Yaskawa INFORM job: pos_z_2.JBI

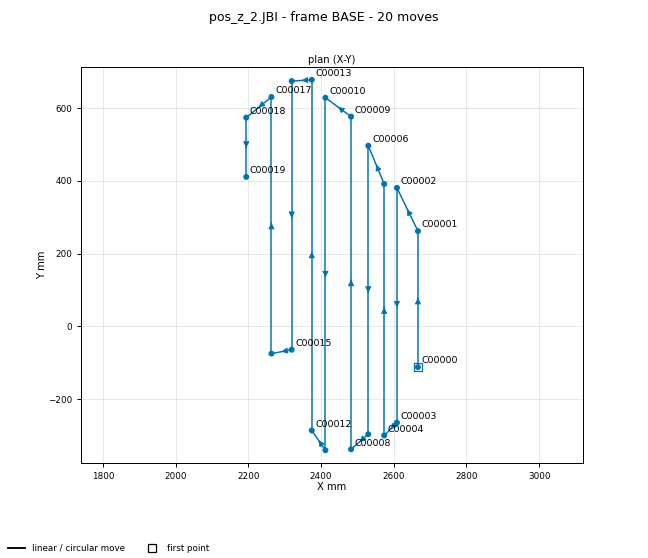
[picture p0: tool path of pos_z_2.JBI in frame BASE, 20 of 22 moves have a stored position in this frame; points joined in program order, loops and branches not executed]
/JOB
//NAME pos_z_2
//POS
///NPOS 20,0,20,0,0,0
///TOOL 0
///POSTYPE BASE
///RECTAN
///RCONF 0,0,0,0,0,0,0,0,0,0,0,0,0,0,0,0,0,0,0,0,0,0,0,0
C00000=2666.772027,-112.261769,-636.738710,-175.000000,-5.000000,-5.000000
C00001=2666.772027,261.995331,-636.738710,-175.000000,-5.000000,-5.000000
C00002=2608.951402,381.030762,-637.876475,-175.000000,-6.408807,-5.000000
C00003=2608.951402,-264.972238,-637.876475,-175.000000,-6.408807,-5.000000
C00004=2573.873265,-300.284116,-636.280803,-175.000000,-5.000000,-5.000000
C00005=2573.873265,391.651884,-636.280803,-175.000000,-5.000000,-5.000000
C00006=2530.108738,496.843725,-636.212429,-175.000000,-5.000000,-5.000000
C00007=2530.108738,-296.777275,-636.212429,-175.000000,-5.000000,-5.000000
C00008=2482.744724,-338.156662,-636.192294,-175.000000,5.000000,5.000000
C00009=2482.744724,577.032338,-636.192294,-175.000000,5.000000,5.000000
C00010=2412.197987,628.980369,-637.311364,-175.000000,-5.483082,-5.000000
C00011=2412.197987,-340.849631,-637.311364,-175.000000,-5.483082,-5.000000
C00012=2374.660605,-286.469165,-636.397181,-175.000000,-5.000000,-5.000000
C00013=2374.660605,678.109835,-636.397181,-175.000000,-5.000000,-5.000000
C00014=2319.427106,674.681551,-636.677680,-175.000000,-5.000000,-5.000000
C00015=2319.427106,-64.307929,-636.677680,-175.000000,-5.000000,-5.000000
C00016=2263.641899,-74.961593,-637.096476,-175.000000,-5.070659,-5.000000
C00017=2263.641899,630.971707,-637.096476,-175.000000,-5.070659,-5.000000
C00018=2194.360285,574.343532,-639.505887,-175.000000,-10.645317,-5.000000
C00019=2194.360285,411.097532,-639.505887,-175.000000,-10.645317,-5.000000
///POSTYPE PULSE
///PULSE
EX000=0
///POSTYPE PULSE
///PULSE
EC00000=0
EC00001=0
EC00002=0
EC00003=0
EC00004=0
EC00005=0
EC00006=0
EC00007=0
EC00008=0
EC00009=0
EC00010=0
EC00011=0
EC00012=0
EC00013=0
EC00014=0
EC00015=0
EC00016=0
EC00017=0
EC00018=0
EC00019=0
//INST
///DATE 2023/06/22 16:21
///ATTR SC,RW,RJ
////FRAME BASE
///GROUP1 RB1,ST1
NOP
MOVJ P009 EX000 VJ=15.00
MOVJ C00000 EC00000 VJ=15.0
CALL JOB:SPYON
MOVL C00001 EC00001 V=150.0
MOVL C00002 EC00002 V=150.0
MOVL C00003 EC00003 V=150.0
MOVL C00004 EC00004 V=150.0
MOVL C00005 EC00005 V=150.0
MOVL C00006 EC00006 V=150.0
MOVL C00007 EC00007 V=150.0
MOVL C00008 EC00008 V=150.0
MOVL C00009 EC00009 V=150.0
MOVL C00010 EC00010 V=150.0
MOVL C00011 EC00011 V=150.0
MOVL C00012 EC00012 V=150.0
MOVL C00013 EC00013 V=150.0
MOVL C00014 EC00014 V=150.0
MOVL C00015 EC00015 V=150.0
MOVL C00016 EC00016 V=150.0
MOVL C00017 EC00017 V=150.0
MOVL C00018 EC00018 V=150.0
MOVL C00019 EC00019 V=150.0
CALL JOB:SPYOF
MOVJ P009 VJ=15.00
END
